FUNCTION_BLOCK FlushFlowSpManager (* Basic Function Block Type *)
  (* Standard: 61499-2 *)
  (* Version 0.0, 7/10/2026, Schneider Electric, Template *)
  PACKAGE SE.Nereda;
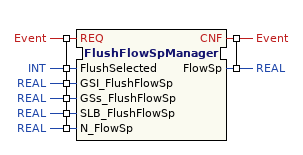
  EVENT_INPUT
    REQ WITH FlushSelected, GSI_FlushFlowSp, GSs_FlushFlowSp, SLB_FlushFlowSp, N_FlowSp; (* Normal Execution Request *)
  END_EVENT
  EVENT_OUTPUT
    CNF WITH FlowSp; (* Execution Confirmation *)
  END_EVENT
  VAR_INPUT
    FlushSelected : INT;
    GSI_FlushFlowSp : REAL;
    GSs_FlushFlowSp : REAL;
    SLB_FlushFlowSp : REAL;
    N_FlowSp : REAL;
  END_VAR
  VAR_OUTPUT
    FlowSp : REAL;
  END_VAR
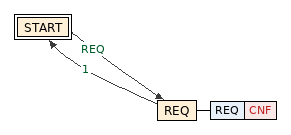
  EC_STATES
    START; (* Initial State *)
    REQ : REQ -> CNF; (* Normal execution *)
  END_STATES
  EC_TRANSITIONS
    START TO REQ := REQ;
    REQ TO START := 1;
  END_TRANSITIONS
  ALGORITHM INIT IN ST: (* Initialization algorithm *)
;
  END_ALGORITHM
  ALGORITHM REQ IN ST: (* Normally executed algorithm *)
;
IF FlushSelected = 0 THEN
	FlowSp := N_FlowSp;
ELSIF FlushSelected = 1 THEN
	FlowSp := GSI_FlushFlowSp;
ELSIF FlushSelected = 2 THEN
	FlowSp := GSs_FlushFlowSp;
ELSIF FlushSelected = 3 THEN
	FlowSp := SLB_FlushFlowSp;
END_IF;
  END_ALGORITHM
END_FUNCTION_BLOCK
